Xinje XCPPro project, PLC1: XC3-24 (software 3.3L)

PROGRAM Ladder

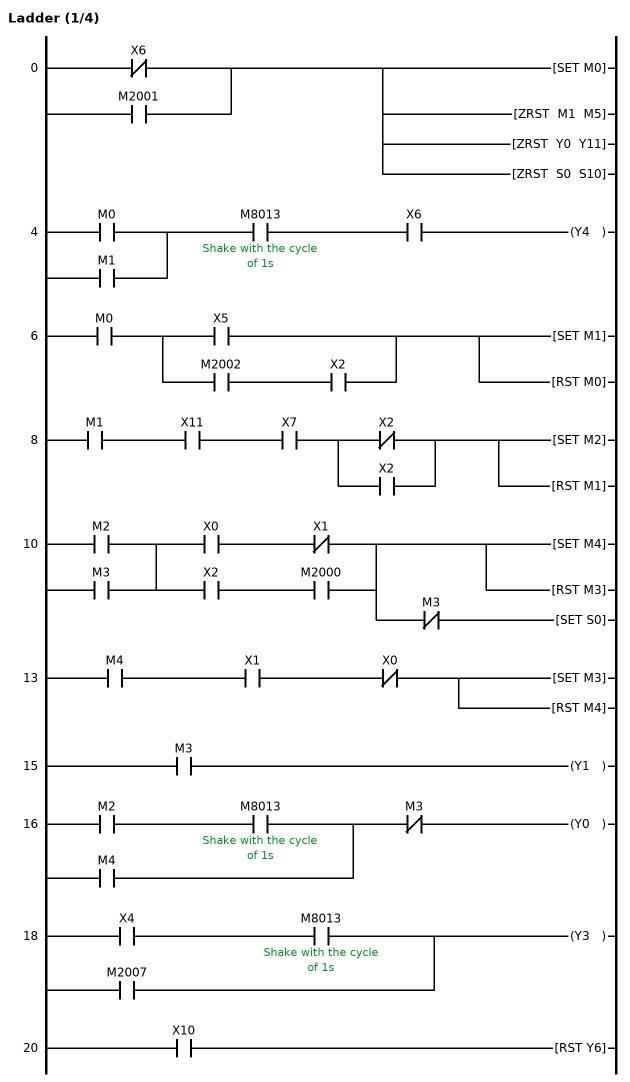
LDI    X6
OR     M2001
SET    M0
ZRST   M1 M5
ZRST   Y0 Y11
ZRST   S0 S10
LD     M0
OR     M1
AND    M8013	; Shake with the cycle of 1s
AND    X6
OUT    Y4
LD     M0
LD     X5
LD     M2002
AND    X2
ORB
ANB
SET    M1
RST    M0
LD     M1
AND    X11
AND    X7
LDI    X2
OR     X2
ANB
SET    M2
RST    M1
LD     M2
OR     M3
LD     X0
ANI    X1
LD     X2
AND    M2000
ORB
ANB
SET    M4
RST    M3
ANI    M3
SET    S0
LD     M4
AND    X1
ANI    X0
SET    M3
RST    M4
LD     M3
OUT    Y1
LD     M2
AND    M8013	; Shake with the cycle of 1s
OR     M4
ANI    M3
OUT    Y0
LD     X4
AND    M8013	; Shake with the cycle of 1s
OR     M2007
OUT    Y3
LD     X10
RST    Y6

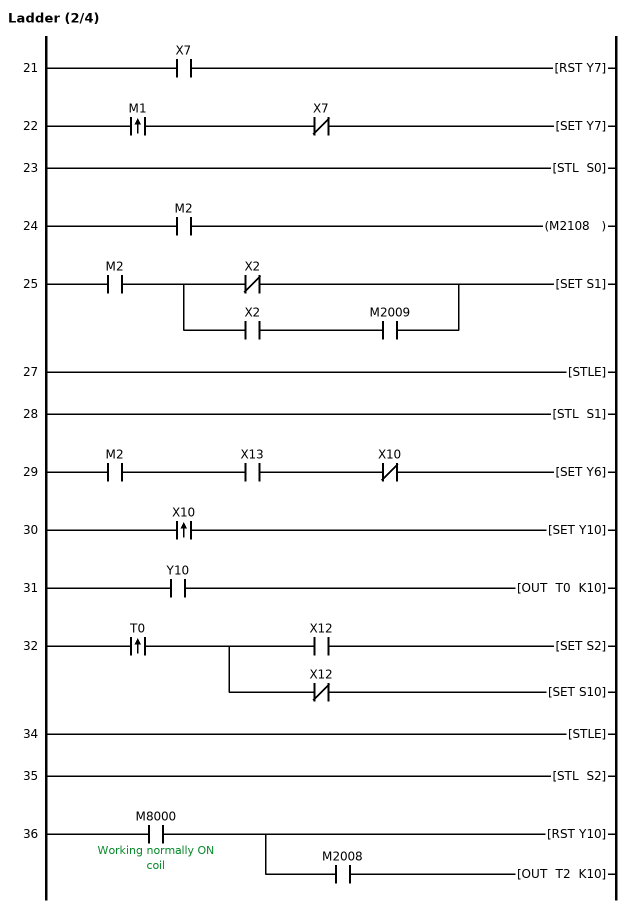
LD     X7
RST    Y7
LDP    M1
ANI    X7
SET    Y7
STL    S0
LD     M2
OUT    M2108
LD     M2
LDI    X2
LD     X2
AND    M2009
ORB
ANB
SET    S1
STLE
STL    S1
LD     M2
AND    X13
ANI    X10
SET    Y6
LDP    X10
SET    Y10
LD     Y10
OUT    T0 K10
LDP    T0
MPS
AND    X12
SET    S2
MPP
ANI    X12
SET    S10
STLE
STL    S2
LD     M8000	; Working normally ON coil
RST    Y10
AND    M2008
OUT    T2 K10

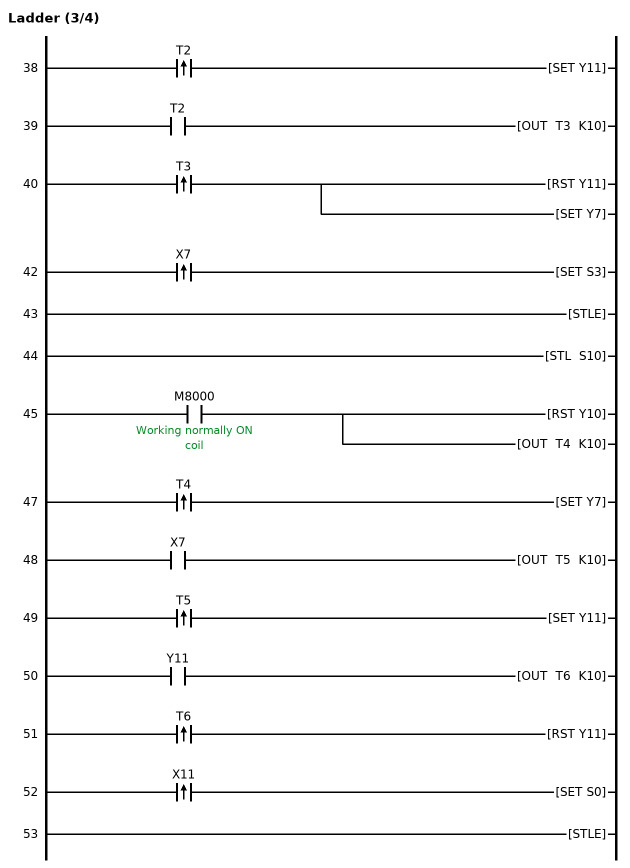
LDP    T2
SET    Y11
LD     T2
OUT    T3 K10
LDP    T3
RST    Y11
SET    Y7
LDP    X7
SET    S3
STLE
STL    S10
LD     M8000	; Working normally ON coil
RST    Y10
OUT    T4 K10
LDP    T4
SET    Y7
LD     X7
OUT    T5 K10
LDP    T5
SET    Y11
LD     Y11
OUT    T6 K10
LDP    T6
RST    Y11
LDP    X11
SET    S0
STLE

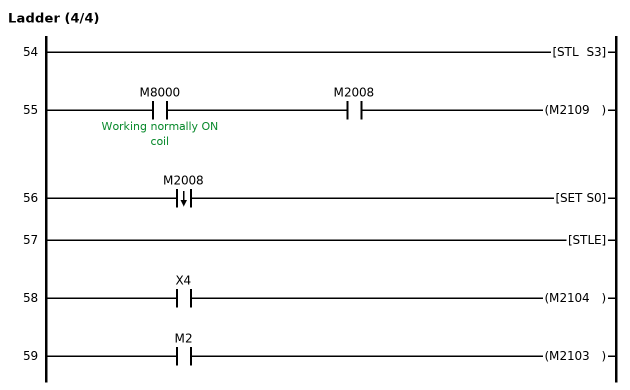
STL    S3
LD     M8000	; Working normally ON coil
AND    M2008
OUT    M2109
LDF    M2008
SET    S0
STLE
LD     X4
OUT    M2104
LD     M2
OUT    M2103